# B&R Automation Studio project lab2
Automation Studio 4.5.2.102

## Configuration SampleText

CPU 4PP065.0571-P74, AutomationRuntime J4.25, Build 4.1.2, Vc V4.25.0, Safety 1.6

### Hardware
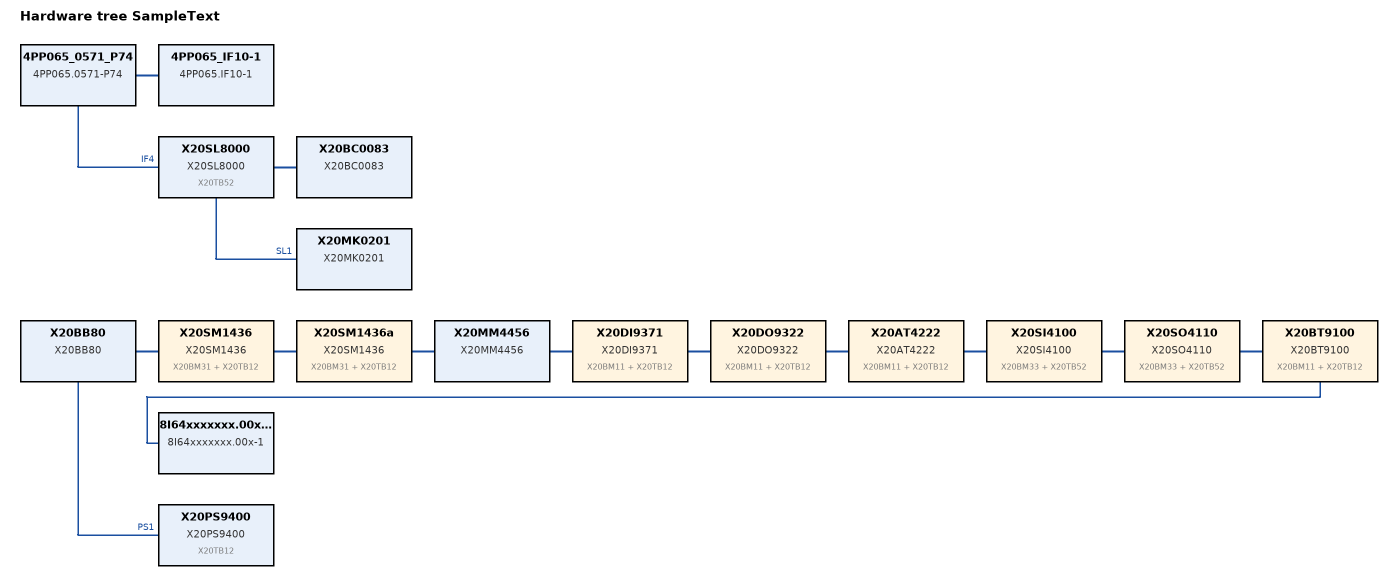
```
4PP065_0571_P74 : 4PP065.0571-P74 v1.1.2.0
  Connector IF4:
    EplInterfaceRedundant = 0
    EplEthInterfaceRedundant = 0
  Connector IF5:
    ActivateDevice = 1
    Mode = Manual
    InternetAddress = 10.1.1.13
    SubnetMask = 255.255.255.0
  ConfigurationID = DriveControl_SampleText
  Simulation = 1
  TimerDeviceType = EPLX2X
  TimerDevice = 4PP065_0571_P74.IF4
  TaskClassIdleTime = 2000
  Cyclic1Duration = 2000
  Cyclic1Tolerance = 0
  Cyclic1Output = 1
4PP065_IF10-1 : 4PP065.IF10-1 v1.0.3.0  [SS -> 4PP065_0571_P74.SS1]
8I64xxxxxxx.00x-1 : 8I64xxxxxxx.00x-1 v1.3.9.1  [X2X1 -> X20BT9100.X2X1 [Cable Type=X2XCable, Length=10, Version=1.0.0.2]]
  packedETAD = packed
  packedETI = packed
  packedCMDD = packed
  packedCMI = packed
  ACC = 30
  DEC = 30
  UNS = 220
  NCR = 10
  NSP = 890
  COS = 64
  RSC = 33000
X20AT4222 : X20AT4222 v1.2.3.0  [SS1 -> X20TB12e.SS; SL -> X20BM11c.SL1]
X20BB80 : X20BB80 v1.0.2.0
X20BC0083 : X20BC0083 v2.7.0.0  [PLK1 -> X20SL8000.PLK2 (NodeNumber=2) [Cable Type=PowerlinkCable, Length=10, Version=1.0.0.2]; SL -> X20BB80.SL1]
X20BM11 : X20BM11 v1.0.0.1  [X2X1 -> X20BM33a.X2X2]
X20BM11a : X20BM11 v1.0.0.1  [X2X1 -> X20MM4456.X2X2]
X20BM11b : X20BM11 v1.0.0.1  [X2X1 -> X20BM11a.X2X2]
X20BM11c : X20BM11 v1.0.0.1  [X2X1 -> X20BM11b.X2X2]
X20BM31 : X20BM31 v1.0.0.1  [X2X1 -> X20BB80.IF1]
X20BM31a : X20BM31 v1.0.0.1  [X2X1 -> X20BM31.X2X2]
X20BM33 : X20BM33 v1.0.0.4  [X2X1 -> X20BM11c.X2X2]
X20BM33a : X20BM33 v1.0.0.4  [X2X1 -> X20BM33.X2X2]
X20BT9100 : X20BT9100 v1.0.3.0  [SS1 -> X20TB12f.SS; SL -> X20BM11.SL1]
X20DI9371 : X20DI9371 v1.0.2.0  [SS1 -> X20TB12c.SS; SL -> X20BM11a.SL1]
X20DO9322 : X20DO9322 v1.0.3.0  [SS1 -> X20TB12d.SS; SL -> X20BM11b.SL1]
X20MK0201 : X20MK0201 v1.0.0.0  [SL -> X20SL8000.SL1]
X20MM4456 : X20MM4456 v1.1.5.0  [X2X1 -> X20BM31a.X2X2]
X20PS9400 : X20PS9400 v1.0.2.4  [SS1 -> X20TB12.SS; PS -> X20BB80.PS1]
X20SI4100 : X20SI4100 v1.10.1.1  [SS1 -> X20TB52.SS; SL -> X20BM33.SL1]
X20SL8000 : X20SL8000 v1.6.5.1  [PLK1 -> 4PP065_0571_P74.IF4 (NodeNumber=1) [Cable Type=PowerlinkCable, Length=10, Version=1.0.0.2]; PLK2 -> X20BC0083.PLK1 (NodeNumber=1) [Cable Type=PowerlinkCable, Length=10, Version=1.0.0.2]; SS1 -> X20TB52b.SS]
  SafeProject = SafeLOGIC-1
X20SM1436 : X20SM1436 v1.4.2.1  [SS1 -> X20TB12a.SS; SL -> X20BM31.SL1]
X20SM1436a : X20SM1436 v1.4.2.1  [SS1 -> X20TB12b.SS; SL -> X20BM31a.SL1]
X20SO4110 : X20SO4110 v1.10.1.1  [SS1 -> X20TB52a.SS; SL -> X20BM33a.SL1]
  SafeModuleID = 3
X20TB12 : X20TB12 v1.0.0.0
X20TB12a : X20TB12 v1.0.0.0
X20TB12b : X20TB12 v1.0.0.0
X20TB12c : X20TB12 v1.0.0.0
X20TB12d : X20TB12 v1.0.0.0
X20TB12e : X20TB12 v1.0.0.0
X20TB12f : X20TB12 v1.0.0.0
X20TB52 : X20TB52 v1.0.0.1
X20TB52a : X20TB52 v1.0.0.1
X20TB52b : X20TB52 v1.0.0.1
```

### IoMap.iom - 4PP065_0571_P74/IoMap.iom
```iecst
VAR_CONFIG
	Cyclic#1.gAxis01_DrvIf.iLifeCnt AT %IB."8I64xxxxxxx.00x-1".SDC_LifeCnt;
	Cyclic#1.gAxis01_DrvIf.iDrvOK AT %IX."8I64xxxxxxx.00x-1".ETAD_Input_Bool_02;
	Cyclic#1.gAxis01_DrvIf.oSetTime AT %QW."8I64xxxxxxx.00x-1".SDC_SetTime;
	Cyclic#1.::Program:DriveStateMashine.speed AT %QW."8I64xxxxxxx.00x-1".LFRD_Output;
	Cyclic#1.gAxis01_DiDoIf.iLifeCntDriveReady AT %IB."8I64xxxxxxx.00x-1".SDC_LifeCnt;
	Cyclic#1.gAxis01_DiDoIf.iLifeCntDriveEnable AT %IB."8I64xxxxxxx.00x-1".SDC_LifeCnt;
	Cyclic#1.gAxis01_DiDoIf.oDriveEnable AT %QX."8I64xxxxxxx.00x-1".CMDD_Output_Bool_00;
	Cyclic#1.gAxis01_ModuleOk AT %QX."8I64xxxxxxx.00x-1".CMDD_Output_Bool_01;
	Cyclic#1.gAxis01_ModuleOk AT %QX."8I64xxxxxxx.00x-1".CMDD_Output_Bool_02;
	Cyclic#1.gAxis01_ModuleOk AT %IX."8I64xxxxxxx.00x-1".ModuleOk;
	Cyclic#1.gAxis01_DiDoIf.oDriveEnable AT %QX."8I64xxxxxxx.00x-1".CMDD_Output_Bool_03;
	Cyclic#1.gAxis01_DiDoIf.iDriveReady AT %IX."8I64xxxxxxx.00x-1".ETAD_Input_Bool_02;
	::Program:DriveStateMashine.state AT %IW."8I64xxxxxxx.00x-1".ETAD_Input;
	::Program:DriveStateMashine.command AT %QW."8I64xxxxxxx.00x-1".CMDD_Output;
	::Program:DoorStateMashine.direction AT %IX."X20DI9371".DigitalInput01;
	::Program:DoorStateMashine.sw1 AT %IX."X20DI9371".DigitalInput02;
	::Program:DoorStateMashine.sw2 AT %IX."X20DI9371".DigitalInput03;
	::Program:DoorStateMashine.sw3 AT %IX."X20DI9371".DigitalInput04;
	::Program:DoorStateMashine.sw4 AT %IX."X20DI9371".DigitalInput05;
	::Program:LedStateMashine.led1 AT %QX."X20DO9322".DigitalOutput02;
	::Program:LedStateMashine.led2 AT %QX."X20DO9322".DigitalOutput03;
	::Program:LedStateMashine.led3 AT %QX."X20DO9322".DigitalOutput04;
	::Program:LedStateMashine.led4 AT %QX."X20DO9322".DigitalOutput05;
END_VAR
```

## Logical view

### Library Logical/Libraries/DriveLib

#### Types.typ
```iecst
TYPE
	DoorStates : 	STRUCT
		ST_INIT : UINT;
		ST_UNKNOWN : UINT;
		ST_OPEN : UINT;
		ST_CLOSE : UINT;
		ST_ACC_POS : UINT;
		ST_ACC_NEG : UINT;
		ST_POS : UINT;
		ST_NEG : UINT;
		ST_DEC_POS : UINT;
		ST_DEC_NEG : UINT;
	END_STRUCT;
END_TYPE
```

#### DriveLib.fun
```iecst
{REDUND_ERROR} {REDUND_UNREPLICABLE} FUNCTION_BLOCK DriveStateMashine (*TODO: Add your comment here*) (*$GROUP=User,$CAT=User,$GROUPICON=User.png,$CATICON=User.png*)
	VAR_INPUT
		state : {REDUND_UNREPLICABLE} UINT;
		enable : {REDUND_UNREPLICABLE} BOOL;
	END_VAR
	VAR_OUTPUT
		command : {REDUND_UNREPLICABLE} UINT;
		speed : {REDUND_UNREPLICABLE} INT;
	END_VAR
END_FUNCTION_BLOCK

{REDUND_ERROR} FUNCTION_BLOCK DoorStateMashine (*TODO: Add your comment here*) (*$GROUP=User,$CAT=User,$GROUPICON=User.png,$CATICON=User.png*)
	VAR_INPUT
		state : {REDUND_UNREPLICABLE} UINT;
		sw1 : {REDUND_UNREPLICABLE} BOOL;
		sw2 : {REDUND_UNREPLICABLE} BOOL;
		sw3 : {REDUND_UNREPLICABLE} BOOL;
		sw4 : {REDUND_UNREPLICABLE} BOOL;
		direction : {REDUND_UNREPLICABLE} BOOL;
	END_VAR
	VAR_OUTPUT
		speed : INT;
	END_VAR
END_FUNCTION_BLOCK

{REDUND_ERROR} {REDUND_UNREPLICABLE} FUNCTION_BLOCK LedStateMashine (*TODO: Add your comment here*) (*$GROUP=User,$CAT=User,$GROUPICON=User.png,$CATICON=User.png*)
	VAR_INPUT
		state : {REDUND_UNREPLICABLE} UINT;
	END_VAR
	VAR_OUTPUT
		led1 : {REDUND_UNREPLICABLE} BOOL;
		led2 : {REDUND_UNREPLICABLE} BOOL;
		led3 : {REDUND_UNREPLICABLE} BOOL;
		led4 : {REDUND_UNREPLICABLE} BOOL;
		timer : {REDUND_UNREPLICABLE} INT;
	END_VAR
END_FUNCTION_BLOCK
```

#### DoorStateMashine.c
```c
#include <bur/plctypes.h>
#ifdef __cplusplus
	extern "C"
	{
#endif
#include "DriveLib.h"
#ifdef __cplusplus
	};
#endif
/* This function block implements state switching for door control */
void DoorStateMashine(struct DoorStateMashine* inst)
{
	switch(inst->state)
	{
		case ST_INIT:
			{
				if(inst->sw1 == 0 && inst->sw2 == 0 && inst->sw3 == 0 && inst->sw4 == 0) inst->state = ST_UNKNOWN;
				break;
			}
		case ST_UNKNOWN:
			{
				if(inst->direction == 0 && inst->sw1 == 0) inst->state = ST_OPEN;
				if(inst->direction == 1 && inst->sw4 == 1) inst->state = ST_CLOSE;
				break;
			}
		case ST_OPEN:
			{
				inst->speed = 0;
				if(inst->direction == 0) inst->state = ST_ACC_POS;
				break;
			}
		case ST_CLOSE:
			{
				inst->speed = 0;
				if(inst->direction == 1) inst->state = ST_ACC_NEG;
				break;
			}
		case ST_ACC_POS:
			{
				inst->speed = 200;
				if(inst->sw2 == 1) inst->state = ST_POS;
				if(inst->direction == 1) inst->state = ST_DEC_NEG;
				break;
			}
		case ST_ACC_NEG:
			{
				inst->speed = -200;
				if(inst->sw3 == 0) inst->state = ST_NEG;
				if(inst->direction == 0) inst->state = ST_DEC_POS;
				break;
			}
		case ST_POS:
			{
				inst->speed = 100;
				if(inst->sw3 == 1) inst->state = ST_DEC_POS;
				if(inst->direction == 1) inst->state = ST_NEG;
				break;
			}
		case ST_NEG:
			{
				inst->speed = -100;
				if(inst->sw3 == 0) inst->state = ST_DEC_NEG;
				if(inst->direction == 0) inst->state = ST_POS;
				break;
			}
		case ST_DEC_POS:
			{
				inst->speed = 100;
				if(inst->sw4 == 1) inst->state = ST_CLOSE;
				break;
			}
		case ST_DEC_NEG:
			{
				inst->speed = -100;
				if(inst->sw4 == 0) inst->state = ST_OPEN;
				break;
			}
	}
}
```

#### DriveStateMashine.c
```c
#include <bur/plctypes.h>
#ifdef __cplusplus
	extern "C"
	{
#endif
#include "DriveLib.h"
#ifdef __cplusplus
	};
#endif
/* This function block implements state switching for motor control */
void DriveStateMashine(struct DriveStateMashine* inst)
{
	if(inst->enable == 0) inst->command = CMD_SHUTDOWN;
	else
	{
		switch(inst->state & 0x6F)
		{
			case ST_DISABLE:
				inst->command = CMD_SHUTDOWN;
				break;
			case ST_SWITCHED_ON:
				inst->command = CMD_SWITCH_ON;
				break;
			case ST_READY:
				inst->command = CMD_ENABLE;
				break;
		}
	}
}
```

#### LedStateMashine.c
```c
#include <bur/plctypes.h>
#ifdef __cplusplus
	extern "C"
	{
#endif
#include "DriveLib.h"
#ifdef __cplusplus
	};
#endif
/* This function block implements state switching to control indicators */
void LedStateMashine(struct LedStateMashine* inst)
{
	switch(inst->state)
	{
		case ST_INIT:
			{
				break;
			}
		case ST_UNKNOWN:
			{
				if(inst->timer%10 == 9)
				{
					inst->led1 = !inst->led1;
					inst->led2 = !inst->led2;
					inst->led3 = !inst->led3;
					inst->led4 = !inst->led4;
				}
				break;
			}
		case ST_OPEN:
			{
				inst->led1 = 0;
				inst->led2 = 0;
				inst->led3 = 0;
				inst->led4 = 0;
				break;
			}
		case ST_CLOSE:
			{
				inst->led1 = 1;
				inst->led2 = 1;
				inst->led3 = 1;
				inst->led4 = 1;
				break;
			}
		case ST_ACC_POS:
			{
				if(inst->timer%10 == 4) inst->led1 = 1;
				inst->led2 = 0;
				inst->led3 = 0;
				inst->led4 = 0;
				break;
			}
		case ST_ACC_NEG:
			{
				inst->led1 = 1;
				inst->led2 = 1;
				inst->led3 = 1;
				if(inst->timer%10 == 4) inst->led4 = 0;
				break;
			}
		case ST_POS:
			{
				inst->led1 = 1;
				if(inst->timer%10 == 9) inst->led2 = 1;
				inst->led3 = 0;
				inst->led4 = 0;
				break;
			}
		case ST_NEG:
			{
				inst->led1 = 1;
				inst->led2 = 1;
				if(inst->timer%10 == 9) inst->led3 = 0;
				inst->led4 = 0;
				break;
			}
		case ST_DEC_POS:
			{
				inst->led1 = 1;
				inst->led2 = 1;
				if(inst->timer%10 == 4) inst->led3 = 1;
				inst->led4 = 0;
				break;
			}
		case ST_DEC_NEG:
			{
				inst->led1 = 1;
				if(inst->timer%10 == 4) inst->led2 = 0;
				inst->led3 = 0;
				inst->led4 = 0;
				break;
			}
	}
}
```

### Program Logical/Program

#### Variables.var
```iecst
VAR
	drive : DriveStateMashine := (0);
	door : DoorStateMashine := (0);
	led : LedStateMashine := (0);
END_VAR
```

#### Main.c
```c
#include <bur/plctypes.h>

#ifdef _DEFAULT_INCLUDES
#include <AsDefault.h>
#endif

void _INIT ProgramInit(void)
{
	drive.enable = 1;
}

void _CYCLIC ProgramCyclic(void)
{
	DoorStateMashine(&door);

	drive.speed = door.speed;
	DriveStateMashine(&drive);

	led.state = door.state;
	LedStateMashine(&led);
	led.timer++;
}

void _EXIT ProgramExit(void)
{

}
```
